INTERFACE IUnsupportedEventHandler EXTENDS IEventHandlerBase

END_INTERFACE

(* stored: Version 1.1.0.1, ProductVersion 3.1.4024.3
   Itf IUnsupportedEventHandler: Id {90e32efe-e6ff-41bd-b867-cb8a8c693c47} *)
